(* IEC 61131-3 sources: bcs-engineering-dsl/language/test/generating/loop_test/expected, 3 files *)

(* ---- LoopsFB_decl.st ---- *)
FUNCTION_BLOCK LoopsFB
VAR_INPUT
    iCount: INT;
END_VAR
VAR_OUTPUT
    oSum: INT;
    oProduct: INT;
END_VAR
VAR
    j: INT;
    tempSum: INT;
    tempProduct: INT;
    i: INT := 0;
END_VAR

(* ---- LoopsFB_impl.st ---- *)
tempSum := 0;
tempProduct := 1;
FOR i := 0 TO 5 BY 1 DO
    tempSum := tempSum + i;
END_FOR;
FOR i := 1 TO iCount BY 1 DO
    tempSum := tempSum + i;
END_FOR;
j := 1;
WHILE j <= iCount DO
    tempProduct := tempProduct * j;
    j := j + 1;
END_WHILE;
oSum := tempSum;
oProduct := tempProduct;

(* ---- MAIN_decl.st ---- *)
PROGRAM MAIN
VAR
    TestLoops_count: INT := 5;
    TestLoops_sum: INT;
    TestLoops_product: INT;
    LoopsFBInstance1: LoopsFB;
END_VAR
